TYPE tDriveInNState1 :
STRUCT
	ReadyToEnable	: BIT;
	Ready			: BIT;
	Warning			: BIT;
	Error			: BIT;
	MovingPositive	: BIT;
	MovingNegative	: BIT;
	TorqueReduced	: BIT;
	Unused			: BIT;
END_STRUCT
END_TYPE

(* stored: Version 1.1.0.1, ProductVersion 3.1.4024.9
   DUT tDriveInNState1: Id {7dd1b971-1990-42a1-a4d1-46458bc8658f} *)
